INTERFACE TrajectoryControllable

PROPERTY ArrivedAtDestination : Bool
GET
END_GET
SET
END_SET
END_PROPERTY

PROPERTY Driving : Bool
GET
END_GET
SET
END_SET
END_PROPERTY

PROPERTY Enable : BOOL
GET
END_GET
SET
END_SET
END_PROPERTY

PROPERTY RobotPose : RobotPose;
GET
END_GET
SET
END_SET
END_PROPERTY

METHOD setWaypointList
VAR_INPUT
	WaypointList : ARRAY[1...30] OF RobotPose;
END_VAR
END_METHOD

PROPERTY WaypointIndex : UINT
GET
END_GET
SET
END_SET
END_PROPERTY

//TODO: define max number of waypoints!
PROPERTY WaypointList : ARRAY[1...30] OF RobotPose
GET
END_GET
SET
END_SET
END_PROPERTY

END_INTERFACE

(* stored: Version 1.1.0.1, ProductVersion 3.1.4024.11
   Itf TrajectoryControllable: Id {90ae884d-3e12-4a80-a4c6-b43944ca7142}
   Property ArrivedAtDestination: Id {941a7901-7b1a-4dca-8745-19d8c1ada202}
   Get Get: Id {b3ff5405-c4df-4e72-a87f-db41b31d1e9b}
   Set Set: Id {e26c7421-edf6-4854-b736-a732583f297a}
   Property Driving: Id {2c0b048d-6a1d-487a-b337-513c2ee62bb4}
   Get Get: Id {10555b5f-fed2-46e8-90e8-dcf121e5c63b}
   Set Set: Id {2423a97d-5afe-4d1a-9678-9bd1f2117bb4}
   Property Enable: Id {4e846c67-ac5f-4f68-8cf5-48b12161e0e0}
   Get Get: Id {8f3d2a89-1085-4b63-9292-29fe81ff55f3}
   Set Set: Id {9ec6ac5a-3552-48ae-a1ad-0dc4b3b81ace}
   Property RobotPose: Id {1f39b865-9249-455a-859e-761edbb87880}
   Get Get: Id {d94aa37a-1574-47ff-8785-2e35884ffe98}
   Set Set: Id {5c954878-14f1-423a-9452-eeca776ef2f5}
   Method setWaypointList: Id {befe7839-4fb2-4598-9c5b-7a386ff7eff2}
   Property WaypointIndex: Id {43bed594-3e20-406a-86bc-725ad6e98b56}
   Get Get: Id {89df4607-ffd7-4057-950a-7f358df67b0c}
   Set Set: Id {09a85252-ec6c-42e6-b87d-ac578880e4b7}
   Property WaypointList: Id {0f714a63-4da7-4ce4-970a-5f548b22afcc}
   Get Get: Id {df97e5eb-b2c4-4a74-b86e-f8c094cde9ee}
   Set Set: Id {6f3d24fe-4b55-4e1d-881a-39f1d07213bf} *)
